TYPE DUT_stProcessingHMIData1 :
STRUCT
	LocationId 			: DINT;
	PartId	 			: DINT;
END_STRUCT
END_TYPE

(* stored: Version 1.1.0.1, ProductVersion 3.1.4024.15
   DUT DUT_stProcessingHMIData1: Id {2e407a49-f4b6-4e6f-8d72-aad213fff784} *)
